PROGRAM d_Mq6

(**-----[4.] MQ6, LPG GAS LEAKAGE DETECTION ---------------------------------------**)
(**LOCAL : Leakage-detected Bit Defined as "bMq6T" **)
IF iMq6 < 6000 THEN
	bMq6T:=FALSE;
ELSIF iMq6 > 6000	THEN
	bMq6T:=TRUE;
END_IF
(**------------------------------------------------**)

(**OUTPUT : Buzzer Output value Defined **)
bMq6latch:=bMq6T OR (bMq6latch AND (NOT bMq6dismiss));
bMq6O:=bMq6latch;
(**-------------------------------------**)
(**------------------------------------------------------------------------------------**)

END_PROGRAM

(* stored: Version 1.1.0.1, ProductVersion 3.1.4018.9
   POU d_Mq6: Id {3f7682e7-5654-418c-960d-d3f7ef8405cf}, SpecialFunc None *)
